TYPE aT_FireCombuster :
STRUCT
	Temperature: LREAL;
END_STRUCT
END_TYPE

(* stored: Version 1.1.0.1, ProductVersion 3.1.4024.4
   DUT aT_FireCombuster: Id {997949e2-45b4-4824-b81d-c947afa2d329} *)
